(* PLC project Tc2_Utilities.FIX16Add Demo, tc3-libraries-kb TwinCAT 3.1 *)
(* stored: creationDateTime 2026-05-10T11:00:00, modificationDateTime 2026-05-10T11:00:00 *)

PROGRAM P_Demo_FIX16Add
  VAR
    bResult : T_FIX16;  (* FIX16Add 的返回值 *)
    bRun : BOOL;  (* 触发一次调用 *)
    a : T_FIX16;  (* 测试用本地变量 *)
    b : T_FIX16;  (* 测试用本地变量 *)
  END_VAR

            // ============================================================
// Tc2_Utilities.FIX16Add 演示程序（FUNCTION）
// ============================================================
// 验证步骤：
//   1. 引用 Tc2_Utilities（及依赖类型所在的库）
//   2. 编译 + 登录
//   3. 强制 bRun := TRUE 一个周期
//   4. 观察 bResult 应为 0.25（=0.5+(-0.25)）
// ============================================================

a := LREAL_TO_FIX16(0.5, 8); b := LREAL_TO_FIX16(-0.25, 8);
IF bRun THEN
    bResult := FIX16Add(a, b);
    bRun := FALSE;
END_IF;

          
END_PROGRAM
